// TIA Portal V19 export
TYPE "C501_STU_DME_TYPIC"
   STRUCT
      VGV_L { ExternalAccessible := 'False'; ExternalVisible := 'False'; ExternalWritable := 'False'} : USInt;   // Vrijgave detectie druk te laag
   END_STRUCT;
END_TYPE
